(* CoDeSys 2.3 library: EmsUdp2Lcc.lib *)
(* Libraries: SysLibSem.lib 7.1.13 17:20:52, Standard.LIB 4.10.05 12:14:46 *)

(* Global variable list: EmsDrv_Global *)
VAR_GLOBAL
    bEmsOK : BOOL;
    bPreEmsOK : BOOL;
    lastEmsBild : INT := -1;

	dwEmsFifoOut: ARRAY[0..255] OF DWORD;
	bEmsFifoOutWrIndex: BYTE;
	bEmsFifoOutRdIndex: BYTE;
	bEmsFifoOutCount:BYTE;
    cntFifoOutFull : DWORD := 0;
    cntFifoOutBusy : DWORD := 0;
    hndFifoOutSema : DWORD := 0;
    cntFifoOutSemaErr : DWORD := 0;
    cntFifoOutSemaIni : DWORD := 0;

	dwEmsFifoIn: ARRAY[0..255] OF DWORD;
	bEmsFifoInWrIndex: BYTE;
	bEmsFifoInRdIndex: BYTE;
	bEmsFifoInCount:BYTE;

	EmsBild:ARRAY [1..30] OF BOOL;
	InEms: DWORD := 0;

    byToggle : BYTE;
END_VAR

VAR_GLOBAL RETAIN PERSISTENT
	bRunWithEMS: BOOL;
    bEnableEmsScaling: BOOL;

    bDummy: BOOL;

	iEmsAktBild:INT;


	rKatzMetRef: REAL;
	rHeigMetRef: REAL;
	rSlewMetRef: REAL;
	rAneoMetRef: REAL;
	rTrimMetRef: REAL;
	rLastMetRef: REAL;
	rSkewMetRef: REAL;
	rTravMetRef: REAL;
	rListMetRef: REAL;
	rKatzMetMax: REAL;
	rHeigMetMax: REAL;
	rSlewMetMax: REAL;
	rAneoMetMax: REAL;
	rTrimMetMax: REAL;
	rLastMetMax: REAL;
	rSkewMetMax: REAL;
	rTravMetMax: REAL;
	rListMetMax: REAL;
	rKatzMetMin: REAL;
	rHeigMetMin: REAL;
	rSlewMetMin: REAL;
	rAneoMetMin: REAL;
	rTrimMetMin: REAL;
	rLastMetMin: REAL;
	rSkewMetMin: REAL;
	rTravMetMin: REAL;
	rListMetMin: REAL;

	diKatzAdc:    DINT;
	diHeigAdc:    DINT;
	diSlewAdc:    DINT;
	diAneoAdc:    DINT;
	diTrimAdc:    DINT;
	diLastAdc:    DINT;
	diSkewAdc:    DINT;
	diTravAdc:    DINT;
	diListAdc:    DINT;
	diKatzAdcMax: DINT;
	diHeigAdcMax: DINT;
	diSlewAdcMax: DINT;
	diAneoAdcMax: DINT;
	diTrimAdcMax: DINT;
	diLastAdcMax: DINT;
	diSkewAdcMax: DINT;
	diTravAdcMax: DINT;
	diListAdcMax: DINT;
	diKatzAdcMin: DINT;
	diHeigAdcMin: DINT;
	diSlewAdcMin: DINT;
	diAneoAdcMin: DINT;
	diTrimAdcMin: DINT;
	diLastAdcMin: DINT;
	diSkewAdcMin: DINT;
	diTravAdcMin: DINT;
	diListAdcMin: DINT;

    StackData:  DWORD;

	bSendToEmsOnlyIfChanged:BOOL:=FALSE;
END_VAR

(* Data type *)
TYPE tEMS_ANEO_DIM:
(
	IBSK_ANEO_KMH       		:=16#0000,  (* Einheit des Windsensors in km/h *)
	IBSK_ANEO_MPH       		:=16#0001,  (* Einheit des Windsensors in mph  *)
	IBSK_ANEO_MS        		:=16#0002   (* Einheit des Windsensors in m/s  *)
);
END_TYPE

(* Data type *)
TYPE tEMS_FLIP:
(
	IBSK_FLIP_WL          			 :=16#01,  (* LB Flipper water side left  (down) *)
	IBSK_FLIP_WR          			 :=16#02,  (* LB Flipper water side right (down) *)
	IBSK_FLIP_LR          			 :=16#04,  (* LB Flipper land  side right (down) *)
	IBSK_FLIP_LL          			 :=16#08   (* LB Flipper land  side left  (down) *)
);
END_TYPE

(* Data type *)
TYPE tEMS_IBSK :
(
	IBSK_STEUER       := 0,         (* DB1 = Checksumme über 4-ByteEinheit, DB2 und DB3 = Steuerbezeichnung *)

	IBSK_KATZ_MET     := 101,       (* Float in Meter  *)   (* Meterwert des Antriebes *)
	IBSK_HEIG_MET     := 102,       (* Float in Meter  *)
	IBSK_SLEW_MET     := 103,       (* Float in Grad   *)
	IBSK_ANEO_MET     := 104,       (* Float in m/s    *)
	IBSK_TRIM_MET     := 105,       (* Float in Grad   *)
	IBSK_LAST_MET     := 106,       (* Float in Tonnen *)
	IBSK_SKEW_MET     := 107,       (* Float in Grad   *)
	IBSK_TRAV_MET     := 108,       (* Float in Meter  *)
	IBSK_LIST_MET     := 109,       (* Float in Grad   *)

	IBSK_KATZ_MET_REF := 111,       (* Float *)  (* Refernzwerte der Antriebes *)
	IBSK_HEIG_MET_REF := 112,       (* Float *)
	IBSK_SLEW_MET_REF := 113,       (* Float *)
	IBSK_ANEO_MET_REF := 114,       (* Float *)
	IBSK_TRIM_MET_REF := 115,       (* Float *)
	IBSK_LAST_MET_REF := 116,       (* Float *)
	IBSK_SKEW_MET_REF := 117,       (* Float *)
	IBSK_TRAV_MET_REF := 118,       (* Float *)
	IBSK_LIST_MET_REF := 119,       (* Float *)

 	IBSK_KATZ_ADC     := 121,       (* Integer in Digit von -4096 bis +4095 *)   (* analogwert des Antriebes *)
	IBSK_HEIG_ADC     := 122,       (* Integer in Digit von -4096 bis +4095 *)
	IBSK_SLEW_ADC     := 123,       (* Integer in Digit von -4096 bis +4095 *)
	IBSK_ANEO_ADC     := 124,       (* Integer in Digit von -4096 bis +4095 *)
	IBSK_TRIM_ADC     := 125,       (* Integer in Digit von -4096 bis +4095 *)
	IBSK_LAST_ADC     := 126,       (* Integer in Digit von -4096 bis +4095 *)
	IBSK_SKEW_ADC     := 127,       (* Integer in Digit von -4096 bis +4095 *)
	IBSK_TRAV_ADC     := 128,       (* Integer in Digit von -4096 bis +4095 *)
	IBSK_LIST_ADC     := 129,       (* Integer in Digit von -4096 bis +4095 *)

	IBSK_NORTH_DIR    := 130,       (* Integer *)   (* Nordrichtung in Grad bezueglich Kran vorne (Boom) *)
	IBSK_KATZ_DIR     := 131,       (* Integer *)   (* Bewegungsrichtung des Antriebes *)
	IBSK_HEIG_DIR     := 132,       (* Integer *)   (* wird noch ignoriert *)
	IBSK_SLEW_DIR     := 133,       (* Integer *)
	IBSK_ANEO_DIR     := 134,       (* Integer *)   (* Windrichtung in Grad bezueglich Kran vorne (Boom) *)
	IBSK_TRIM_DIR     := 135,       (* Integer *)
	IBSK_LAST_DIR     := 136,       (* Integer *)
	IBSK_SKEW_DIR     := 137,       (* Integer *)
	IBSK_TRAV_DIR     := 138,       (* Integer *)
	IBSK_LIST_DIR     := 139,       (* Integer *)

	IBSK_STEU_EIN     := 140,       (* Integer 1=An, 0=Aus *)   (* für Maschinendatenerfassung *)
	IBSK_KATZ_EIN     := 141,       (* Integer 1=An, 0=Aus *)
	IBSK_HEIG_EIN     := 142,       (* Integer 1=An, 0=Aus *)
	IBSK_SLEW_EIN     := 143,       (* Integer 1=An, 0=Aus *)
	IBSK_TRIM_EIN     := 145,       (* Integer 1=An, 0=Aus *)
	IBSK_SKEW_EIN     := 147,       (* Integer 1=An, 0=Aus *)
	IBSK_TRAV_EIN     := 148,       (* Integer 1=An, 0=Aus *)
	IBSK_LIST_EIN     := 149,       (* Integer 1=An, 0=Aus *)

	IBSK_KATZ_MET_MAX := 151,       (* Float in Meter  *)
	IBSK_HEIG_MET_MAX := 152,       (* Float in Meter  *)
	IBSK_SLEW_MET_MAX := 153,       (* Float in Grad   *)
	IBSK_ANEO_MET_MAX := 154,       (* Float in m/s    *)
	IBSK_TRIM_MET_MAX := 155,       (* Float in Grad   *)
	IBSK_LAST_MET_MAX := 156,       (* Float in Tonnen *)
	IBSK_SKEW_MET_MAX := 157,       (* Float in Grad   *)
	IBSK_TRAV_MET_MAX := 158,       (* Float in Meter  *)
	IBSK_LIST_MET_MAX := 159,       (* Float in Grad   *)

	IBSK_KATZ_MET_MIN := 161,       (* Float in Meter  *)
	IBSK_HEIG_MET_MIN := 162,       (* Float in Meter  *)
	IBSK_SLEW_MET_MIN := 163,       (* Float in Grad   *)
	IBSK_ANEO_MET_MIN := 164,       (* Float in m/s    *)
	IBSK_TRIM_MET_MIN := 165,       (* Float in Grad   *)
	IBSK_LAST_MET_MIN := 166,       (* Float in Tonnen *)
	IBSK_SKEW_MET_MIN := 167,       (* Float in Grad   *)
	IBSK_TRAV_MET_MIN := 168,       (* Float in Meter  *)
	IBSK_LIST_MET_MIN := 169,       (* Float in Grad   *)

	IBSK_KATZ_ADC_MAX := 171,       (* Integer in digit von -4096 bis 4095 *)
	IBSK_HEIG_ADC_MAX := 172,       (* Integer *)
	IBSK_SLEW_ADC_MAX := 173,       (* Integer *)
	IBSK_ANEO_ADC_MAX := 174,       (* Integer *)
	IBSK_TRIM_ADC_MAX := 175,       (* Integer *)
	IBSK_LAST_ADC_MAX := 176,       (* Integer *)
	IBSK_SKEW_ADC_MAX := 177,       (* Integer *)
	IBSK_TRAV_ADC_MAX := 178,       (* Integer *)
	IBSK_LIST_ADC_MAX := 179,       (* Integer *)

	IBSK_KATZ_ADC_MIN := 181,       (* Integer in digit von -4096 bis 4095 *)
	IBSK_HEIG_ADC_MIN := 182,       (* Integer in digit *)
	IBSK_SLEW_ADC_MIN := 183,       (* Integer in digit *)
	IBSK_ANEO_ADC_MIN := 184,       (* Integer in digit *)
	IBSK_TRIM_ADC_MIN := 185,       (* Integer in digit *)
	IBSK_LAST_ADC_MIN := 186,       (* Integer in digit *)
	IBSK_SKEW_ADC_MIN := 187,       (* Integer in digit *)
	IBSK_TRAV_ADC_MIN := 188,       (* Integer in digit *)
	IBSK_LIST_ADC_MIN := 189,       (* Integer in digit *)

	IBSK_BOOM_INFO    := 196,       (* Integer mit Bitbeutung *)
                                    (* 16#0001 = YES "LS1 Boom Up Activated"  *)
                                    (* 16#0002 = YES "LS2 Boom Up Activated"  *)
                                    (* 16#0004 = YES "Slack Rope Left"        *)
                                    (* 16#0008 = YES "Slack Rope Right"       *)
                                    (* 16#0010 = YES "Hook Open"              *)
                                    (* 16#0020 = YES "Hook Closed"            *)
                                    (* 16#0040 = YES "Boom Locked"            *)
                                    (* 16#0080 = YES "LS > 70° Boom Position" *)
                                    (* 16#0100 = YES "In Locking Zone"        *)
                                    (* 16#0200 = YES "LS Boom Down Activated" *)

	IBSK_BOOM_MET  	  := 197,       (* Float in Grad *)
	IBSK_SPRE_MET     := 198,       (* Float in feet *)

	IBSK_FLIP_TWIN    := 199,       (* Integer LB = Flipper und HB = Twin-Lift *)

                                    (* Funktionsbeschreibung am Spreadder *)
                                    (* FLIP = flipper    *)
                                    (* TWIN = twin-lift  *)
                                    (* LOCK = twist-lock *)
                                    (* PROB = probe-pin = deposition point *)

                                    (* Positionsbeschreibung am Spreadder *)
                                    (* zuert water- oder land-side *)
                                    (* dann left oder right *)
                                    (* w = water side *)
                                    (* l = land  side *)
                                    (* l = left       *)
                                    (* r = right      *)
                                    (* t = twin lift  *)


	IBSK_LOCK_PROB    := 200,       (* Integer twist locks und probe pin *)



	IBSK_ANEO_EINHEIT := 201,       (* Integer *) (* Einheit für den Windsensor *)

	IBSK_X_POS        := 204,       (* Integer *) (* Containerposition *)
	IBSK_Y_POS        := 205,       (* Integer *) (* Containerposition *)
	IBSK_Z_POS        := 206,       (* Integer *) (* Containerposition *)
	IBSK_X_DIR        := 207,       (* Zeichen *) (* +,-,* (entspricht: 1,2,3) *)
	IBSK_Y_DIR        := 208,       (* Zeichen *) (* +,-,* (entspricht: 1,2,3) *)
	IBSK_Z_DIR        := 209,       (* Zeichen *) (* +,-,* (entspricht: 1,2,3) *)

	IBSK_ERROR_SET    := 210,       (* Integer Fehler  setzten *)
	IBSK_ERROR_CLEAR  := 211,       (* Integer Fehler  löschen *)
	IBSK_WARN_SET     := 212,       (* Integer Warnung setzten *)
	IBSK_WARN_CLEAR   := 213,       (* Integer Warnung löschen *)

    IBSK_SPRE2_MET    := 215,       (* Tandemspreader Spreader 2: Float in feet *)
    IBSK_FLIP2_TWIN2  := 216,       (* Tandemspreader Spreader 2: Integer LB = Flipper und HB = Twin-Lift *)
    IBSK_LOCK2_PROB2  := 217,       (* Tandemspreader Spreader 2: Integer twist locks und probe pin *)

	IBSK_BILD         := 220,       (* Integer Bildnummer *)
                                    (*  1 = BILD1                        *)
                                    (*  2 = BILD2                        *)
                                    (*  3 = BILD3                        *)
                                    (*  4 = BILD4                        *)
                                    (*  5 = SCALierbild                  *)
                                    (*  6 = Menübild                     *)
                                    (* 10 = COM2-Testbild                *)
                                    (* 11 = Maschinendatenbild 1         *)
                                    (* 12 = Maschinendatenbild 2         *)
                                    (* 13 = Maschinendatenbild 3         *)
                                    (* 14 = Langzeitmaschinendatenbild 1 *)
                                    (* 15 = Langzeitmaschinendatenbild 2 *)
                                    (* 16 = Langzeitmaschinendatenbild 3 *)
                                    (* 19 = zuletzt angewähltes Bild     *)
                                    (*      der Bilder 1 bis 6           *)
                                    (* 26 = BILD neu zeichnen            *)
                                    (* 27 = IBS-Testbild                 *)
                                    (* 28 = BILD5                        *)
                                    (* 29 = BILD6                        *)
                                    (* 30 = BILD_BOOM                    *)

	IBSK_TAST         := 221,       (* Integer HB = Taste  *)
                                    (* TAS_B4 =  1 *)
                                    (* TAS_CL =  2 *)
                                    (* TAS_B5 =  3 *)
                                    (* TAS_EN =  4 *)
                                    (* TAS_B6 =  5 *)
                                    (* TAS_KE =  6 *)
                                    (* TAS_B7 =  7 *)
                                    (* TAS_LI =  9 *)
                                    (* TAS_B1 = 10 *)
                                    (* TAS_RE = 11 *)
                                    (* TAS_B2 = 12 *)
                                    (* TAS_HO = 13 *)
                                    (* TAS_B3 = 14 *)
                                    (* TAS_AB = 15 *)
                                    (*        LB = Repeat *)
                                    (* 1 <= Repeat <= 255 *)
	IBSK_NEW_COM_MODE := 230,	    (* Integer Umschalten in neuen Kommunikationsmode *)
									(* keine Wandlung von Floats *)
							    	(* Schreiben zum EMS: Daten bleiben stehen, bis neue Daten gesendet werden *)
									(* Lesen von EMS: Auswertung von Daten nur bei Änderung *)

    IBSK_STACK_DATA   := 231,       (* Stackdaten DWORD (4 BYTE) *)
                                    (* -> IBS-Kennung, Daten-Kennung, Stack-Nr, Wert *)

    IBSK_MDE2_DATA    := 232,       (* Maschinendaten Bild2 DWORD (4 BYTE) *)
                                    (* -> IBS-Kennung, Daten-Kennung, WORD-Wert *)
    IBSK_MDE3_DATA    := 233,       (* Maschinendaten Bild3 DWORD (4 BYTE) *)
                                    (* -> IBS-Kennung, Daten-Kennung, WORD-Wert *)

	IBSK_GPS_DELTAY   := 234,		(* Abweichung des Krans von der Stackfahrspur *)
	IBSK_GPS_ANGLE    := 235,		(* Winkel des Krans gegenüber der Stackfahrspur *)
	IBSK_GPS_STEERDIR := 236,		(* Lenkrichtung, um zurück auf did Stackfahrspur zu kommen *)

    IBSK_EMS_MODE     := 237        (* EMS-Modus ; Spezielle/Kundenspezifische Anpassungen *)
                                    (* z.Zt.: 0x01 - IBSK_EMS_MODE_MASK_XYZ_2CHAR *) (* 12.01.04 V2.50        *)
                                    (*        0x02 - IBSK_EMS_MODE_MASK_B3_CUST1  *) (* 12.01.04 V2.50        *)
                                    (*        0x04 - IBSK_EMS_MODE_MASK_YZ_2CHAR  *) (* 13.03.09 V2.55 IR1745 *)
                                    (*        0x08 - IBSK_EMS_MODE_MASK_STACK_BIN *) (* 17.02.11 V2.56 RT188  *)
                                    (*        0x80 - IBSK_EMS_MODE_MASK_SET       *)

);
END_TYPE

(* Data type *)
TYPE tEMS_LOCK:
(
	IBSK_LOCK_WL          		 :=16#01,  (* LB Twist lock           water side left  (locked)  *)
	IBSK_LOCK_WR          		 :=16#02,  (* LB Twist lock           water side right (locked)  *)
	IBSK_LOCK_LR          		 :=16#04,  (* LB Twist lock           land  side left  (locked)  *)
	IBSK_LOCK_LL          		 :=16#08,  (* LB Twist lock           land  side right (locked)  *)
	IBSK_LOCK_TWL         		 :=16#10,  (* LB Twist lock twin lift water side left  (locked)  *)
	IBSK_LOCK_TWR         		 :=16#20,  (* LB Twist lock twin lift water side right (locked)  *)
	IBSK_LOCK_TLR         		 :=16#40,  (* LB Twist lock twin lift land  side left  (locked)  *)
	IBSK_LOCK_TLL         		 :=16#80   (* LB Twist lock twin lift land  side right (locked)  *)
);
END_TYPE

(* Data type *)
TYPE tEMS_MDE2 :
(
	IBSK_MDE2K_UNDEF :=0,    (* Undefiniert *)

	IBSK_MDE2K_STEU_AN_1,    (* Kurzzeitspeicher Steuerung An (Anzahl)   1. WORD *)
	IBSK_MDE2K_STEU_AN_2,    (* Kurzzeitspeicher Steuerung An (Anzahl)   2. WORD *)
	IBSK_MDE2K_STEU_ZEIT_1,  (* Kurzzeitspeicher Steuerung An (Dauer)    1. WORD *)
	IBSK_MDE2K_STEU_ZEIT_2,  (* Kurzzeitspeicher Steuerung An (Dauer)    2. WORD *)
	IBSK_MDE2K_KATZ_AN_1,    (* Kurzzeitspeicher Katzantrieb An (Anzahl) 1. WORD *)
	IBSK_MDE2K_KATZ_AN_2,    (* Kurzzeitspeicher Katzantrieb An (Anzahl) 2. WORD *)
	IBSK_MDE2K_KATZ_ZEIT_1,  (* Kurzzeitspeicher Katzantrieb An (Dauer)  1. WORD *)
	IBSK_MDE2K_KATZ_ZEIT_2,  (* Kurzzeitspeicher Katzantrieb An (Dauer)  2. WORD *)
	IBSK_MDE2K_DREH_AN_1,    (* Kurzzeitspeicher Drehantrieb An (Anzahl) 1. WORD *)
	IBSK_MDE2K_DREH_AN_2,    (* Kurzzeitspeicher Drehantrieb An (Anzahl) 2. WORD *)
	IBSK_MDE2K_DREH_ZEIT_1,  (* Kurzzeitspeicher Drehantrieb An (Dauer)  1. WORD *)
	IBSK_MDE2K_DREH_ZEIT_2,  (* Kurzzeitspeicher Drehantrieb An (Dauer)  2. WORD *)
	IBSK_MDE2K_HUB_AN_1,     (* Kurzzeitspeicher Hubantrieb An (Anzahl)  1. WORD *)
	IBSK_MDE2K_HUB_AN_2,     (* Kurzzeitspeicher Hubantrieb An (Anzahl)  2. WORD *)
	IBSK_MDE2K_HUB_ZEIT_1,   (* Kurzzeitspeicher Hubantrieb An (Dauer)   1. WORD *)
	IBSK_MDE2K_HUB_ZEIT_2,   (* Kurzzeitspeicher Hubantrieb An (Dauer)   2. WORD *)
	IBSK_MDE2K_FAHR_AN_1,    (* Kurzzeitspeicher Fahrantrieb An (Anzahl) 1. WORD *)
	IBSK_MDE2K_FAHR_AN_2,    (* Kurzzeitspeicher Fahrantrieb An (Anzahl) 2. WORD *)
	IBSK_MDE2K_FAHR_ZEIT_1,  (* Kurzzeitspeicher Fahrantrieb An (Dauer)  1. WORD *)
	IBSK_MDE2K_FAHR_ZEIT_2,  (* Kurzzeitspeicher Fahrantrieb An (Dauer)  2. WORD *)

	IBSK_MDE2L_STEU_AN_1,    (* Langzeitspeicher Steuerung An (Anzahl)   1. WORD *)
	IBSK_MDE2L_STEU_AN_2,    (* Langzeitspeicher Steuerung An (Anzahl)   2. WORD *)
	IBSK_MDE2L_STEU_ZEIT_1,  (* Langzeitspeicher Steuerung An (Dauer)    1. WORD *)
	IBSK_MDE2L_STEU_ZEIT_2,  (* Langzeitspeicher Steuerung An (Dauer)    2. WORD *)
	IBSK_MDE2L_KATZ_AN_1,    (* Langzeitspeicher Katzantrieb An (Anzahl) 1. WORD *)
	IBSK_MDE2L_KATZ_AN_2,    (* Langzeitspeicher Katzantrieb An (Anzahl) 2. WORD *)
	IBSK_MDE2L_KATZ_ZEIT_1,  (* Langzeitspeicher Katzantrieb An (Dauer)  1. WORD *)
	IBSK_MDE2L_KATZ_ZEIT_2,  (* Langzeitspeicher Katzantrieb An (Dauer)  2. WORD *)
	IBSK_MDE2L_DREH_AN_1,    (* Langzeitspeicher Drehantrieb An (Anzahl) 1. WORD *)
	IBSK_MDE2L_DREH_AN_2,    (* Langzeitspeicher Drehantrieb An (Anzahl) 2. WORD *)
	IBSK_MDE2L_DREH_ZEIT_1,  (* Langzeitspeicher Drehantrieb An (Dauer)  1. WORD *)
	IBSK_MDE2L_DREH_ZEIT_2,  (* Langzeitspeicher Drehantrieb An (Dauer)  2. WORD *)
	IBSK_MDE2L_HUB_AN_1,     (* Langzeitspeicher Hubantrieb An (Anzahl)  1. WORD *)
	IBSK_MDE2L_HUB_AN_2,     (* Langzeitspeicher Hubantrieb An (Anzahl)  2. WORD *)
	IBSK_MDE2L_HUB_ZEIT_1,   (* Langzeitspeicher Hubantrieb An (Dauer)   1. WORD *)
	IBSK_MDE2L_HUB_ZEIT_2,   (* Langzeitspeicher Hubantrieb An (Dauer)   2. WORD *)
	IBSK_MDE2L_FAHR_AN_1,    (* Langzeitspeicher Fahrantrieb An (Anzahl) 1. WORD *)
	IBSK_MDE2L_FAHR_AN_2,    (* Langzeitspeicher Fahrantrieb An (Anzahl) 2. WORD *)
	IBSK_MDE2L_FAHR_ZEIT_1,  (* Langzeitspeicher Fahrantrieb An (Dauer)  1. WORD *)
	IBSK_MDE2L_FAHR_ZEIT_2,  (* Langzeitspeicher Fahrantrieb An (Dauer)  2. WORD *)

	IBSK_MDE2K_LOESCH_1,     (* Kurzzeitspeicher letzte Loeschzeit       1. WORD *)
	IBSK_MDE2K_LOESCH_2,     (* Kurzzeitspeicher letzte Loeschzeit       2. WORD *)

	IBSK_MDE2L_LOESCH_1,     (* Langzeitspeicher letzte Loeschzeit       1. WORD *)
	IBSK_MDE2L_LOESCH_2      (* Langzeitspeicher letzte Loeschzeit       2. WORD *)
);
END_TYPE

(* Data type *)
TYPE tEMS_MDE3 :
(
	IBSK_MDE3K_UNDEF :=0,    (* Undefiniert *)

	IBSK_MDE3K_BIS10_1,      (* Kurzzeitspeicher Last bis 10%       1. WORD *)
	IBSK_MDE3K_BIS10_2,      (* Kurzzeitspeicher Last bis 10%       2. WORD *)
	IBSK_MDE3K_BIS33_1,      (* Kurzzeitspeicher Last bis 33%       1. WORD *)
	IBSK_MDE3K_BIS33_2,      (* Kurzzeitspeicher Last bis 33%       2. WORD *)
	IBSK_MDE3K_BIS66_1,      (* Kurzzeitspeicher Last bis 66%       1. WORD *)
	IBSK_MDE3K_BIS66_2,      (* Kurzzeitspeicher Last bis 66%       2. WORD *)
	IBSK_MDE3K_BIS100_1,     (* Kurzzeitspeicher Last bis 100%      1. WORD *)
	IBSK_MDE3K_BIS100_2,     (* Kurzzeitspeicher Last bis 100%      2. WORD *)
	IBSK_MDE3K_AB100_1,      (* Kurzzeitspeicher Last ueber 100%    1. WORD *)
	IBSK_MDE3K_AB100_2,      (* Kurzzeitspeicher Last ueber 100%    2. WORD *)

	IBSK_MDE3L_BIS10_1,      (* Langzeitspeicher Last bis 10%       1. WORD *)
	IBSK_MDE3L_BIS10_2,      (* Langzeitspeicher Last bis 10%       2. WORD *)
	IBSK_MDE3L_BIS33_1,      (* Langzeitspeicher Last bis 33%       1. WORD *)
	IBSK_MDE3L_BIS33_2,      (* Langzeitspeicher Last bis 33%       2. WORD *)
	IBSK_MDE3L_BIS66_1,      (* Langzeitspeicher Last bis 66%       1. WORD *)
	IBSK_MDE3L_BIS66_2,      (* Langzeitspeicher Last bis 66%       2. WORD *)
	IBSK_MDE3L_BIS100_1,     (* Langzeitspeicher Last bis 100%      1. WORD *)
	IBSK_MDE3L_BIS100_2,     (* Langzeitspeicher Last bis 100%      2. WORD *)
	IBSK_MDE3L_AB100_1,      (* Langzeitspeicher Last ueber 100%    1. WORD *)
	IBSK_MDE3L_AB100_2,      (* Langzeitspeicher Last ueber 100%    2. WORD *)

	IBSK_MDE3K_LOESCH_1,     (* Kurzzeitspeicher letzte Loeschzeit  1. WORD *)
	IBSK_MDE3K_LOESCH_2,     (* Kurzzeitspeicher letzte Loeschzeit  2. WORD *)

	IBSK_MDE3L_LOESCH_1,     (* Langzeitspeicher letzte Loeschzeit  1. WORD *)
	IBSK_MDE3L_LOESCH_2      (* Langzeitspeicher letzte Loeschzeit  2. WORD *)
);
END_TYPE

(* Data type *)
TYPE tEMS_MODE :
(
  (* EMS-Modus ; Spezielle/Kundenspezifische Anpassungen (fuer Interbuskennung IBSK_EMS_MODE := 237) *)
  IBSK_EMS_MODE_MASK_SET       := 16#80,  (* EMS_MODE_MASK_... gesetzt *)
  IBSK_EMS_MODE_MASK_XYZ_2CHAR := 16#01,  (* 12.01.04 V2.50        *)
  IBSK_EMS_MODE_MASK_B3_CUST1  := 16#02,  (* 12.01.04 V2.50        *)
  IBSK_EMS_MODE_MASK_YZ_2CHAR  := 16#04,  (* 13.03.09 V2.55 IR1745 *)
  IBSK_EMS_MODE_MASK_STACK_BIN := 16#08   (* 17.02.11 V2.56 RT188  *)
);
END_TYPE

(* Data type *)
TYPE tEMS_PROBE:
(
	IBSK_PROB_WL          		 :=16#01,  (* HB Probe pin            water side left  (pressed) *)
	IBSK_PROB_WR          		 :=16#02,  (* HB Probe pin            water side right (pressed) *)
	IBSK_PROB_LR          		 :=16#04,  (* HB Probe pin            land  side left  (pressed) *)
	IBSK_PROB_LL          		 :=16#08,  (* HB Probe pin            land  side right (pressed) *)
	IBSK_PROB_TWL         		 :=16#10,  (* HB Probe pin  twin lift water side left  (pressed) *)
	IBSK_PROB_TWR         		 :=16#20,  (* HB Probe pin  twin lift water side right (pressed) *)
	IBSK_PROB_TLR         		 :=16#40,  (* HB Probe pin  twin lift land  side left  (pressed) *)
	IBSK_PROB_TLL         		 :=16#80   (* HB Probe pin  twin lift land  side right (pressed) *)
);
END_TYPE

(* Data type *)
TYPE tEMS_STACK :
(
	IBSK_STACK_UNDEF :=0,  (* Undefiniert *)
	IBSK_STACK_SIZEX,      (* Stacklaenge Travel in 10ft-Einheiten *)
	IBSK_STACK_SIZEY,      (* Stackbreite Trolley in Container-Einheiten *)
	IBSK_STACK_SIZEZ,      (* Stacklaenge Hoist in Container-Einheiten *)
	IBSK_STACK_AKTNR,      (* Aktuelle Stacknummer *)
	IBSK_STACK_NAME0,      (* Stackname 1. Char *)
	IBSK_STACK_NAME1,      (* Stackname 2. Char *)
	IBSK_STACK_DIRROW,     (* Stackausrichtung  Row - Trolley *)
	IBSK_STACK_LABELY,     (* Bezeichnung der Stack-Y-Richtung *)
	IBSK_STACK_FIRST,      (* Position des ersten Containers speichern *)
	IBSK_STACK_LAST,       (* Position des letzten Containers speichern *)
    IBSK_STACK_LABELZ,     (* Bezeichnung der Stack-Z-Richtung *)
	IBSK_STACK_DIRCOL,     (* Stackausrichtung  Column - Travel *)
    IBSK_STACK_FIRST_X1,   (* 1. BYTE des float-Werts der X-Position des ersten Containers *)
    IBSK_STACK_FIRST_X2,   (* 2. BYTE des float-Werts der X-Position des ersten Containers *)
    IBSK_STACK_FIRST_X3,   (* 3. BYTE des float-Werts der X-Position des ersten Containers *)
    IBSK_STACK_FIRST_Y1,   (* 1. BYTE des float-Werts der Y-Position des ersten Containers *)
    IBSK_STACK_FIRST_Y2,   (* 2. BYTE des float-Werts der Y-Position des ersten Containers *)
    IBSK_STACK_FIRST_Y3,   (* 3. BYTE des float-Werts der Y-Position des ersten Containers *)
    IBSK_STACK_LAST_X1,    (* 1. BYTE des float-Werts der X-Position des letzten Containers *)
    IBSK_STACK_LAST_X2,    (* 2. BYTE des float-Werts der X-Position des letzten Containers *)
    IBSK_STACK_LAST_X3,    (* 3. BYTE des float-Werts der X-Position des letzten Containers *)
    IBSK_STACK_LAST_Y1,    (* 1. BYTE des float-Werts der Y-Position des letzten Containers *)
    IBSK_STACK_LAST_Y2,    (* 2. BYTE des float-Werts der Y-Position des letzten Containers *)
    IBSK_STACK_LAST_Y3,    (* 3. BYTE des float-Werts der Y-Position des letzten Containers *)
    IBSK_STACK_AKT_X1,     (* 1. BYTE des float-Werts der aktuellen X-Position *)
    IBSK_STACK_AKT_X2,     (* 2. BYTE des float-Werts der aktuellen X-Position *)
    IBSK_STACK_AKT_X3,     (* 3. BYTE des float-Werts der aktuellen X-Position *)
    IBSK_STACK_AKT_Y1,     (* 1. BYTE des float-Werts der aktuellen Y-Position *)
    IBSK_STACK_AKT_Y2,     (* 2. BYTE des float-Werts der aktuellen Y-Position *)
    IBSK_STACK_AKT_Y3      (* 3. BYTE des float-Werts der aktuellen Y-Position *)
);
END_TYPE

(* Data type *)
TYPE tEMS_STACK_DATA :
STRUCT
 kenn   : tEMS_STACK;
 nr     : BYTE;
 data   : BYTE;
 toggle : BYTE;
END_STRUCT
END_TYPE

(* Data type *)
TYPE tEMS_TWIN :
(
	IBSK_TWIN             			 :=16#01,  (* HB Twin-lift (aktiv) *)
	IBSK_TANDEM            			 :=16#02,  (* HB Twin-lift (aktiv) *)
	IBSK_ENABLED           			 :=16#04   (* HB Twin-lift (aktiv) *)
);
END_TYPE

(* POU BoomInfoToEms, ST *)
PROGRAM BoomInfoToEms
VAR_INPUT
	Ls1BoomUpActivated: BOOL;
	Ls2BoomUpActivated: BOOL;
	SlackRopeLeft: BOOL;
	SlackRopeRight: BOOL;
	HookOpen: BOOL;
	HookClosed: BOOL;
	BoomLocked: BOOL;
	LsGreater70DegBoomPosition: BOOL;

	InLockingZone: BOOL;
	LsBoomDownActivated: BOOL;
END_VAR
VAR
	pdw: POINTER TO ARRAY[0..3] OF BYTE;
	dwEMSOut: DWORD := 0;
END_VAR
pdw := ADR(dwEMSOut);

pdw^[0] := INT_TO_BYTE(IBSK_LOCK_PROB);
(*pdw^[1] := 0;*)
pdw^[1] := byToggle;
byToggle := byToggle + 1;

pdw^[2].0 := InLockingZone;
pdw^[2].1 := LsBoomDownActivated;


pdw^[3].0 := Ls1BoomUpActivated;
pdw^[3].1 := Ls2BoomUpActivated;
pdw^[3].2 := SlackRopeLeft;
pdw^[3].3 := SlackRopeRight;
pdw^[3].4 := HookOpen;
pdw^[3].5 := HookClosed;
pdw^[3].6 := BoomLocked;
pdw^[3].7 := LsGreater70DegBoomPosition;

EmsOutFifo(dwEMSOut);
END_PROGRAM

(* POU EmsOutFifo, ST *)
FUNCTION EmsOutFifo : BOOL
VAR_INPUT
	dwEmsOut:DWORD;
END_VAR
VAR
 bSemRet : BOOL;
END_VAR
IF( hndFifoOutSema > 0) THEN
 bSemRet := SysSemEnter( hndFifoOutSema);
 IF( bSemRet) THEN

  (* noch Platz im Fifo ?*)
  (*IF (bEmsFifoOutCount <= 255) THEN*)
  IF( bEmsFifoOutCount < 255) THEN
   (*ins Fifo schreiben*)
   dwEmsFifoOut[bEmsFifoOutWrIndex] := dwEmsOut;
   bEmsFifoOutWrIndex := bEmsFifoOutWrIndex+1;
   bEmsFifoOutCount := bEmsFifoOutCount+1;
   EmsOutFifo:=TRUE;
  ELSE
   cntFifoOutFull := cntFifoOutFull + 1;
   EmsOutFifo:=FALSE;
  END_IF

  bSemRet := SysSemLeave( hndFifoOutSema);
  IF( NOT bSemRet) THEN
   cntFifoOutSemaErr := cntFifoOutSemaErr + 1;
  END_IF
 ELSE
  cntFifoOutBusy := cntFifoOutBusy + 1;
 END_IF
ELSE
 cntFifoOutSemaIni := cntFifoOutSemaIni + 1;
END_IF
END_FUNCTION

(* POU EMS_BildUpdate, ST *)
PROGRAM EMS_BildUpdate
VAR
	ii:BYTE;
END_VAR
(* beim Erststart auf Bild1 umschalten *)
IF (iEmsAktBild = -1) THEN
	BildNumToEms(1);

ELSE
	FOR ii:=1 TO 30 BY 1 DO
		IF (EmsBild[ii] = TRUE) THEN
			BildNumToEms(ii);
		END_IF
	END_FOR
END_IF
END_PROGRAM

(* POU BildNumToEms, ST *)
FUNCTION BildNumToEms:BOOL
VAR_INPUT
	Wert: INT;
END_VAR
VAR
	pdw: POINTER TO ARRAY[0..3] OF BYTE;
	pint: POINTER TO ARRAY[0..1] OF BYTE;
	dwEMSOut: DWORD;
END_VAR
pdw := ADR(dwEMSOut);
pint := ADR(Wert);

pdw^[0] := INT_TO_BYTE(IBSK_BILD);
(*pdw^[1] := 0;*)
pdw^[1] := byToggle;
byToggle := byToggle + 1;
pdw^[2] := pint^[1];
pdw^[3] := pint^[0];

BildNumToEms := EmsOutFifo(dwEMSOut);
END_FUNCTION

(* POU EMS_DataInterpreter, ST *)
PROGRAM EMS_DataInterpreter
VAR_INPUT
	bEnable: BOOL;
END_VAR
VAR
	dwEmsIn:DWORD;
	Kennung:tEMS_IBSK;
END_VAR
IF NOT bEnable THEN
	RETURN;
END_IF

IF (bEmsFifoInCount > 0) THEN
	(*aus Fifo lesen *)
	dwEmsIn := dwEmsFifoIn[bEmsFifoInRdIndex];
	bEmsFifoInRdIndex := bEmsFifoInRdIndex+1;
	bEmsFifoInCount := bEmsFifoInCount-1;
	Kennung := GetIbsKennung(dwEmsIn);

	CASE Kennung OF
		IBSK_STEUER:
	;
		IBSK_KATZ_MET,	(* Float in Meter  *)   (* Meterwert des Antriebes *)
		IBSK_HEIG_MET,  (* Float in Meter  *)
		IBSK_SLEW_MET,  (* Float in Grad   *)
		IBSK_ANEO_MET,  (* Float in m/s    *)
		IBSK_TRIM_MET,  (* Float in Grad   *)
		IBSK_LAST_MET,  (* Float in Tonnen *)
		IBSK_SKEW_MET,  (* Float in Grad   *)
		IBSK_TRAV_MET,  (* Float in Meter  *)
		IBSK_LIST_MET:  (* Float in Grad   *)
	;
		IBSK_KATZ_MET_REF:  (* Float *)  (* Refernzwerte der Antriebes *)
			rKatzMetRef := FloatFromEms(dwEmsIn);
		IBSK_HEIG_MET_REF:  (* Float *)
			rHeigMetRef := FloatFromEms(dwEmsIn);
		IBSK_SLEW_MET_REF:  (* Float *)
			rSlewMetRef := FloatFromEms(dwEmsIn);
		IBSK_ANEO_MET_REF:  (* Float *)
			rAneoMetRef := FloatFromEms(dwEmsIn);
		IBSK_TRIM_MET_REF:  (* Float *)
			rTrimMetRef := FloatFromEms(dwEmsIn);
		IBSK_LAST_MET_REF:  (* Float *)
			rLastMetRef := FloatFromEms(dwEmsIn);
		IBSK_SKEW_MET_REF:  (* Float *)
			rSkewMetRef := FloatFromEms(dwEmsIn);
		IBSK_TRAV_MET_REF:  (* Float *)
			rTravMetRef := FloatFromEms(dwEmsIn);
		IBSK_LIST_MET_REF:  (* Float *)
			rListMetRef := FloatFromEms(dwEmsIn);


		IBSK_KATZ_MET_MAX:  (* Float in Meter  *)
			rKatzMetMax := FloatFromEms(dwEmsIn);
		IBSK_HEIG_MET_MAX:  (* Float in Meter  *)
			rHeigMetMax := FloatFromEms(dwEmsIn);
		IBSK_SLEW_MET_MAX:  (* Float in Grad   *)
			rSlewMetMax := FloatFromEms(dwEmsIn);
		IBSK_ANEO_MET_MAX:  (* Float in m/s    *)
			rAneoMetMax := FloatFromEms(dwEmsIn);
		IBSK_TRIM_MET_MAX:  (* Float in Grad   *)
			rTrimMetMax := FloatFromEms(dwEmsIn);
		IBSK_LAST_MET_MAX: (* Float in Tonnen *)
			rLastMetMax := FloatFromEms(dwEmsIn);
		IBSK_SKEW_MET_MAX:  (* Float in Grad   *)
			rSkewMetMax := FloatFromEms(dwEmsIn);
		IBSK_TRAV_MET_MAX:  (* Float in Meter  *)
			rTravMetMax := FloatFromEms(dwEmsIn);
		IBSK_LIST_MET_MAX:  (* Float in Grad   *)
			rListMetMax := FloatFromEms(dwEmsIn);

		IBSK_KATZ_MET_MIN:  (* Float in Meter  *)
			rKatzMetMin := FloatFromEms(dwEmsIn);
		IBSK_HEIG_MET_MIN:  (* Float in Meter  *)
			rHeigMetMin := FloatFromEms(dwEmsIn);
		IBSK_SLEW_MET_MIN:  (* Float in Grad   *)
			rSlewMetMin := FloatFromEms(dwEmsIn);
		IBSK_ANEO_MET_MIN:  (* Float in m/s    *)
			rAneoMetMin := FloatFromEms(dwEmsIn);
		IBSK_TRIM_MET_MIN:  (* Float in Grad   *)
			rTrimMetMin := FloatFromEms(dwEmsIn);
		IBSK_LAST_MET_MIN:  (* Float in Tonnen *)
			rLastMetMin := FloatFromEms(dwEmsIn);
		IBSK_SKEW_MET_MIN:  (* Float in Grad   *)
			rSkewMetMin := FloatFromEms(dwEmsIn);
		IBSK_TRAV_MET_MIN:  (* Float in Meter  *)
			rTravMetMin := FloatFromEms(dwEmsIn);
		IBSK_LIST_MET_MIN:  (* Float in Grad   *)
			rListMetMin := FloatFromEms(dwEmsIn);

	 	IBSK_KATZ_ADC:			(* Integer in Digit von -4096 bis +4095 *)   (* analogwert des Antriebes *)
			diKatzAdc := IntFromEms(dwEmsIn);
		IBSK_HEIG_ADC:  		(* Integer in Digit von -4096 bis +4095 *)
			diHeigAdc := IntFromEms(dwEmsIn);
		IBSK_SLEW_ADC:  		(* Integer in Digit von -4096 bis +4095 *)
			diSlewAdc := IntFromEms(dwEmsIn);
		IBSK_ANEO_ADC:  		(* Integer in Digit von -4096 bis +4095 *)
			diAneoAdc := IntFromEms(dwEmsIn);
		IBSK_TRIM_ADC:			(* Integer in Digit von -4096 bis +4095 *)
			diTrimAdc := IntFromEms(dwEmsIn);
		IBSK_LAST_ADC:  (* Integer in Digit von -4096 bis +4095 *)
			diLastAdc := IntFromEms(dwEmsIn);
		IBSK_SKEW_ADC:  (* Integer in Digit von -4096 bis +4095 *)
			diSkewAdc := IntFromEms(dwEmsIn);
		IBSK_TRAV_ADC:  (* Integer in Digit von -4096 bis +4095 *)
			diTravAdc := IntFromEms(dwEmsIn);
		IBSK_LIST_ADC:  (* Integer in Digit von -4096 bis +4095 *)
			diListAdc := IntFromEms(dwEmsIn);

		IBSK_KATZ_DIR,  (* Integer *)   (* Bewegungsrichtung des Antriebes *)
		IBSK_HEIG_DIR,  (* Integer *)   (* wird noch ignoriert *)
		IBSK_SLEW_DIR,  (* Integer *)
		IBSK_ANEO_DIR,  (* Integer *)
		IBSK_TRIM_DIR,  (* Integer *)
		IBSK_LAST_DIR,  (* Integer *)
		IBSK_SKEW_DIR,  (* Integer *)
		IBSK_TRAV_DIR,  (* Integer *)
		IBSK_LIST_DIR: (* Integer *)
	;
		IBSK_STEU_EIN,  (* Integer 1=An, 0=Aus *)   (* für Maschinendatenerfassung *)
		IBSK_KATZ_EIN,  (* Integer 1=An, 0=Aus *)
		IBSK_HEIG_EIN,  (* Integer 1=An, 0=Aus *)
		IBSK_SLEW_EIN,  (* Integer 1=An, 0=Aus *)
		IBSK_TRIM_EIN,  (* Integer 1=An, 0=Aus *)
		IBSK_SKEW_EIN,  (* Integer 1=An, 0=Aus *)
		IBSK_TRAV_EIN,  (* Integer 1=An, 0=Aus *)
		IBSK_LIST_EIN:  (* Integer 1=An, 0=Aus *)
	;

		IBSK_KATZ_ADC_MAX:  (* Integer in digit von -4096 bis 4095 *)
			diKatzAdcMax := IntFromEms(dwEmsIn);
		IBSK_HEIG_ADC_MAX:  (* Integer *)
			diHeigAdcMax := IntFromEms(dwEmsIn);
		IBSK_SLEW_ADC_MAX:  (* Integer *)
			diSlewAdcMax := IntFromEms(dwEmsIn);
		IBSK_ANEO_ADC_MAX:  (* Integer *)
			diAneoAdcMax := IntFromEms(dwEmsIn);
		IBSK_TRIM_ADC_MAX:  (* Integer *)
			diTrimAdcMax := IntFromEms(dwEmsIn);
		IBSK_LAST_ADC_MAX:  (* Integer *)
			diLastAdcMax := IntFromEms(dwEmsIn);
		IBSK_SKEW_ADC_MAX:  (* Integer *)
			diSkewAdcMax := IntFromEms(dwEmsIn);
		IBSK_TRAV_ADC_MAX:  (* Integer *)
			diTravAdcMax := IntFromEms(dwEmsIn);
		IBSK_LIST_ADC_MAX: (* Integer *)
			diListAdcMax := IntFromEms(dwEmsIn);

		IBSK_KATZ_ADC_MIN:  (* Integer in digit von -4096 bis 4095 *)
			diKatzAdcMin := IntFromEms(dwEmsIn);
		IBSK_HEIG_ADC_MIN:  (* Integer in digit *)
			diHeigAdcMin := IntFromEms(dwEmsIn);
		IBSK_SLEW_ADC_MIN:  (* Integer in digit *)
			diSlewAdcMin := IntFromEms(dwEmsIn);
		IBSK_ANEO_ADC_MIN:  (* Integer in digit *)
			diAneoAdcMin := IntFromEms(dwEmsIn);
		IBSK_TRIM_ADC_MIN:  (* Integer in digit *)
			diTrimAdcMin := IntFromEms(dwEmsIn);
		IBSK_LAST_ADC_MIN:  (* Integer in digit *)
			diLastAdcMin := IntFromEms(dwEmsIn);
		IBSK_SKEW_ADC_MIN:  (* Integer in digit *)
			diSkewAdcMin := IntFromEms(dwEmsIn);
		IBSK_TRAV_ADC_MIN:  (* Integer in digit *)
			diTravAdcMin := IntFromEms(dwEmsIn);
		IBSK_LIST_ADC_MIN:  (* Integer in digit *)
			diListAdcMin := IntFromEms(dwEmsIn);

		IBSK_BOOM_INFO:  (* Integer mit Bitbeutung *)
	                                 (* 16#0001 = YES "LS1 Boom Up Activated"  *)
	                                 (* 16#0002 = YES "LS2 Boom Up Activated"  *)
	                                 (* 16#0004 = YES "Slack Rope Left"        *)
	                                 (* 16#0008 = YES "Slack Rope Right"       *)
	                                 (* 16#0010 = YES "Hook Open"              *)
	                                 (* 16#0020 = YES "Hook Closed"            *)
	                                 (* 16#0040 = YES "Boom Locked"            *)
	                                 (* 16#0080 = YES "LS > 70° Boom Position" *)
	                                 (* 16#0100 = YES "In Locking Zone"        *)
	                                 (* 16#0200 = YES "LS Boom Down Activated" *)
	;
		IBSK_BOOM_MET,  (* Float in Grad *)
		IBSK_SPRE_MET:  (* Float in feet *)
	;
		IBSK_FLIP_TWIN:  (* Integer LB = Flipper und HB = Twin-Lift *)
	;
	                                 (* Funktionsbeschreibung am Spreadder *)
	                                 (* FLIP = flipper    *)
	                                 (* TWIN = twin-lift  *)
	                                 (* LOCK = twist-lock *)
	                                 (* PROB = probe-pin = deposition point *)

	                                    (* Positionsbeschreibung am Spreadder *)
	                                    (* zuert water- oder land-side *)
	                                    (* dann left oder right *)
	                                    (* w = water side *)
	                                    (* l = land  side *)
	                                    (* l = left       *)
	                                    (* r = right      *)
	                                    (* t = twin lift  *)


		IBSK_LOCK_PROB:  (* Integer twist locks und probe pin *)
	;


		IBSK_ANEO_EINHEIT:  (* Integer *) (* Einheit für den Windsensor *)
	;
		IBSK_X_POS,  (* Integer *) (* Containerposition *)
		IBSK_Y_POS,  (* Integer *) (* Containerposition *)
		IBSK_Z_POS,  (* Integer *) (* Containerposition *)
		IBSK_X_DIR,  (* Zeichen *) (* +,-,* *)
		IBSK_Y_DIR,  (* Zeichen *) (* +,-,* *)
		IBSK_Z_DIR:  (* Zeichen *) (* +,-,* *)
	;
		IBSK_ERROR_SET:    (* Integer Fehler  setzten *)
	;
		IBSK_ERROR_CLEAR:  (* Integer Fehler  löschen *)
	;
		IBSK_WARN_SET:     (* Integer Warnung setzten *)
	;
		IBSK_WARN_CLEAR:   (* Integer Warnung löschen *)
	;
		IBSK_BILD: (* Integer Bildnummer *)
			iEmsAktBild := INT_TO_BYTE(IntFromEms(dwEmsIn));
		IBSK_TAST:  (* Integer HB = Taste  *)
	;                                   (* TAS_B4 =  1 *)
	                                    (* TAS_CL =  2 *)
	                                    (* TAS_B5 =  3 *)
	                                    (* TAS_EN =  4 *)
	                                    (* TAS_B6 =  5 *)
	                                    (* TAS_KE =  6 *)
	                                    (* TAS_B7 =  7 *)
	                                    (* TAS_LI =  9 *)
	                                    (* TAS_B1 = 10 *)
	                                    (* TAS_RE = 11 *)
	                                    (* TAS_B2 = 12 *)
	                                    (* TAS_HO = 13 *)
	                                    (* TAS_B3 = 14 *)
	                                    (* TAS_AB = 15 *)
	                                    (*        LB = Repeat *)
	                                    (* 1 <= Repeat <= 255 *)

        IBSK_STACK_DATA:                (* Stackdaten DWORD (4 Byte) *)
            StackData := dwEmsIn;

	END_CASE
END_IF
END_PROGRAM

(* POU GetIbsKennung, ST *)
FUNCTION GetIbsKennung : tEMS_IBSK
VAR_INPUT
	InEMS:DWORD;
END_VAR
VAR
	pdw: POINTER TO ARRAY[0..3] OF BYTE;
END_VAR
pdw := ADR(InEMS);
GetIbsKennung := pdw^[0];
END_FUNCTION

(* POU FloatFromEms, ST *)
FUNCTION FloatFromEms:REAL
VAR_INPUT
	dwEMSIn: DWORD;
END_VAR
VAR
	pdw		: POINTER TO ARRAY[0..3] OF BYTE;
	pWert	: POINTER TO ARRAY[0..3] OF BYTE;
	Wert: REAL;
END_VAR
pdw := ADR(dwEMSIn);
pWert := ADR(Wert);

(* ibs   = mmmmmmmm emmmmmmm seeeeeee kkkkkkkk *)
(* float = seeeeeee emmmmmmm mmmmmmmm mmmmmmmm *)

(* Wert füllen und dabei Bytereihenfolge drehen *)
pWert^[0] := 0;
pWert^[1] := pdw^[3];
pWert^[2] := pdw^[2];
pWert^[3] := pdw^[1];

FloatFromEms := Wert;
END_FUNCTION

(* POU IntFromEms, ST *)
FUNCTION IntFromEms: INT
VAR_INPUT
	dwEMSIn: DWORD;
END_VAR
VAR
	pdw: POINTER TO ARRAY[0..3] OF BYTE;
	pint: POINTER TO ARRAY[0..1] OF BYTE;

	Kennung: tEMS_IBSK;
	Wert: INT;
END_VAR
pdw := ADR(dwEMSIn);
pint := ADR(Wert);

Kennung := pdw^[0];
pint^[1] := pdw^[2];
pint^[0] := pdw^[3];

IntFromEms := Wert;
END_FUNCTION

(* POU EMS_Init, ST *)
PROGRAM EMS_Init

VAR_INPUT
	bEnable:BOOL;
END_VAR

VAR
	bRestart: BOOL := TRUE;
	rtEnable: R_TRIG;
	fbIntToEms:IntToEms;
	Wert:INT;

	Counter: BYTE;
	ton1s: TON;
END_VAR
IF( hndFifoOutSema = 0) THEN
 hndFifoOutSema := SysSemCreate( TRUE);
END_IF

rtEnable( CLK := bEnable);

IF rtEnable.Q THEN
  (* clear FifoOut *)
  bEmsFifoOutCount := 0;
  bEmsFifoOutRdIndex := 0;
  bEmsFifoOutWrIndex := 0;
  (* send New Mode to EMS in both dwords *)
  Counter := 0;
END_IF

ton1s( IN := TRUE, PT := t#1s);

IF ( ton1s.Q = TRUE) AND ( Counter < 5) THEN
  fbIntToEms( Kennung := IBSK_NEW_COM_MODE, Wert := Wert);
  Counter := Counter + 1;
  ton1s( IN := FALSE);
END_IF
END_PROGRAM

(* POU IntToEms, ST *)
FUNCTION_BLOCK IntToEms
VAR_INPUT
	Kennung: tEMS_IBSK;
	Wert: INT;
END_VAR
VAR
	pdw: POINTER TO ARRAY[0..3] OF BYTE;
	pint: POINTER TO ARRAY[0..1] OF BYTE;
	dwEMSOut: DWORD;
	LastdwEMSOut: DWORD;
END_VAR
pdw := ADR(dwEMSOut);
pint := ADR(Wert);

pdw^[0] := INT_TO_BYTE(Kennung);
(*pdw^[1] := 0;*)
pdw^[1] := byToggle;
byToggle := byToggle + 1;
pdw^[2] := pint^[1];
pdw^[3] := pint^[0];

IF bSendToEmsOnlyIfChanged THEN
	IF (LastdwEMSOut <> dwEMSOut) THEN
		EmsOutFifo(dwEMSOut);
	END_IF
ELSE
	EmsOutFifo(dwEMSOut);
END_IF
LastdwEMSOut := dwEMSOut;
END_FUNCTION_BLOCK

(* POU EMS_Mode, ST *)
PROGRAM EMS_Mode

VAR_INPUT
  bEnable : BOOL;
  iWert   : INT;
END_VAR

VAR
  rtEnable : R_TRIG;
  fbIntToEms : IntToEms;

  Counter : BYTE;
  ton1s : TON;
END_VAR
rtEnable( CLK := bEnable);

IF rtEnable.Q THEN
  (* send EMS mode to EMS every second for 5 seconds *)
  Counter := 0;
END_IF

ton1s( IN := TRUE, PT := t#1s);

IF ( ton1s.Q = TRUE) AND ( Counter < 5) THEN
  fbIntToEms( Kennung := IBSK_EMS_MODE, Wert := iWert);
  Counter := Counter + 1;
  ton1s( IN := FALSE);
END_IF
END_PROGRAM

(* POU EMS_Read, ST *)
PROGRAM EMS_Read
VAR_INPUT
	bEnable: BOOL;
	In1: DWORD;
	In2: DWORD;
END_VAR
VAR
	idwEms1Old:DWORD:=0;
	idwEms2Old:DWORD:=0;
END_VAR
IF NOT bEnable OR NOT bRunWithEMS THEN
	RETURN;
END_IF

(* EMS-Daten einlesen *)
IF (In1<>idwEms1Old) THEN
	EmsInFifo(In1);
	idwEms1Old:=In1;
END_IF
IF (In2<>idwEms2Old) THEN
	EmsInFifo(In2);
	idwEms2Old:=In2;
END_IF
END_PROGRAM

(* POU EmsInFifo, ST *)
FUNCTION EmsInFifo : BOOL
VAR_INPUT
	dwEmsIn:DWORD;
END_VAR
VAR
END_VAR
(* noch Platz im Fifo ?*)
IF (bEmsFifoInCount <= 255) THEN
	(*ins Fifo schreiben*)
	 dwEmsFifoIn[bEmsFifoInWrIndex] := dwEmsIn;
	bEmsFifoInWrIndex := bEmsFifoInWrIndex+1;
	bEmsFifoInCount := bEmsFifoInCount+1;
  EmsInFifo:=TRUE;
ELSE
  EmsInFifo:=FALSE;
END_IF
END_FUNCTION

(* POU EMS_Write, ST *)
PROGRAM EMS_Write
VAR_INPUT
  bEnable: BOOL;
END_VAR
VAR_OUTPUT
  Out1: DWORD;
  Out2: DWORD;
END_VAR
VAR
  rtEnable: R_TRIG;
  LastChannel: BYTE := 1;
  bSemRet : BOOL;
END_VAR
rtEnable(CLK:=bEnable);
IF (rtEnable.Q) THEN
	LastChannel := 2;
END_IF

IF NOT bEnable OR NOT bRunWithEMS THEN
	RETURN;
END_IF


IF( hndFifoOutSema > 0) THEN
 bSemRet := SysSemEnter( hndFifoOutSema);
 IF( bSemRet) THEN

  IF (bEmsFifoOutCount>0) THEN
	(* FifoOut-Daten zum EMS senden *)
	IF(LastChannel = 1) THEN
		LastChannel := 2;
	ELSE
		LastChannel := 1;
	END_IF
	IF(LastChannel = 1) THEN
		Out1 := dwEmsFifoOut[bEmsFifoOutRdIndex];
	ELSE
		Out2 := dwEmsFifoOut[bEmsFifoOutRdIndex];
	END_IF
	bEmsFifoOutRdIndex := bEmsFifoOutRdIndex+1;
	bEmsFifoOutCount := bEmsFifoOutCount-1;
  END_IF

  bSemRet := SysSemLeave( hndFifoOutSema);
  IF( NOT bSemRet) THEN
   cntFifoOutSemaErr := cntFifoOutSemaErr + 1;
  END_IF
 ELSE
  cntFifoOutBusy := cntFifoOutBusy + 1;
 END_IF
ELSE
 cntFifoOutSemaIni := cntFifoOutSemaIni + 1;
END_IF
END_PROGRAM

(* POU FlipTwinToEms, ST *)
PROGRAM FlipTwinToEms
VAR_INPUT
	FlipWaterSideLeftDown: BOOL;
	FlipWaterSideRightDown: BOOL;
	FlipLandSideRightDown: BOOL;
	FlipLandSideLeftDown: BOOL;
	TwinLiftActive: BOOL;
END_VAR
VAR_OUTPUT
    FlippersToEMS : WORD;
    TwinToEMS : WORD;
END_VAR
TwinToEMS.0 := TwinLiftActive;

FlippersToEMS.0 := FlipWaterSideLeftDown;
FlippersToEMS.1 := FlipWaterSideRightDown;
FlippersToEMS.2 := FlipLandSideRightDown;
FlippersToEMS.3 := FlipLandSideLeftDown;
END_PROGRAM

(* POU LockProbToEms, ST *)
PROGRAM LockProbToEms
VAR_INPUT
	TlWaterSideLeftLocked: BOOL;
	TlWaterSideRightLocked: BOOL;
	TlLandSideLeftLocked: BOOL;
	TlLandSideRightLocked: BOOL;
	TlTwinLiftWaterSideLeftLocked: BOOL;
	TlTwinLiftWaterSideRightLocked: BOOL;
	TlTwinLiftLandSideLeftLocked: BOOL;
	TlTwinLiftLandSideRightLocked: BOOL;

	PpWaterSideLeftPressed: BOOL;
	PpWaterSideRightPressed: BOOL;
	PpLandSideLeftPressed: BOOL;
	PpLandSideRightPressed: BOOL;
	PpTwinLiftWaterSideLeftPressed: BOOL;
	PpTwinLiftWaterSideRightPressed: BOOL;
	PpTwinLiftLandSideLeftPressed: BOOL;
	PpTwinLiftLandSideRightPressed: BOOL;
END_VAR
VAR_OUTPUT
    TwistlocksToEMS : WORD;
    ProbesToEMS : WORD;
END_VAR
ProbesToEMS.0 := PpWaterSideLeftPressed;
ProbesToEMS.1 := PpWaterSideRightPressed;
ProbesToEMS.2 := PpLandSideRightPressed;
ProbesToEMS.3 := PpLandSideLeftPressed;
ProbesToEMS.4 := PpTwinLiftWaterSideLeftPressed;
ProbesToEMS.5 := PpTwinLiftWaterSideRightPressed;
ProbesToEMS.6 := PpTwinLiftLandSideRightPressed;
ProbesToEMS.7 := PpTwinLiftLandSideLeftPressed;


TwistlocksToEMS.0 := TlWaterSideLeftLocked;
TwistlocksToEMS.1 := TlWaterSideRightLocked;
TwistlocksToEMS.2 := TlLandSideRightLocked;
TwistlocksToEMS.3 := TlLandSideLeftLocked;
TwistlocksToEMS.4 := TlTwinLiftWaterSideLeftLocked;
TwistlocksToEMS.5 := TlTwinLiftWaterSideRightLocked;
TwistlocksToEMS.6 := TlTwinLiftLandSideRightLocked;
TwistlocksToEMS.7 := TlTwinLiftLandSideLeftLocked;
END_PROGRAM

(* POU BuildStackData, ST *)
FUNCTION BuildStackData : tEMS_STACK_DATA
VAR_INPUT
 kenn : tEMS_STACK;
 nr   : BYTE;
 data : BYTE;
END_VAR
VAR
END_VAR
BuildStackData.kenn := kenn;
BuildStackData.nr := nr;
BuildStackData.data := data;
END_FUNCTION

(* POU DirToEms, ST *)
FUNCTION_BLOCK DirToEms
VAR_INPUT
	Kennung: tEMS_IBSK;
	Wert: STRING;
END_VAR
VAR
	pdw: POINTER TO ARRAY[0..3] OF BYTE;
	dwEMSOut: DWORD;
	LastdwEMSOut: DWORD;
END_VAR
(*
Wert: '+' (1) 
Wert: '-' (2)
Wert: '*' (3)
*)
pdw := ADR(dwEMSOut);

pdw^[0] := INT_TO_BYTE(Kennung);
(*pdw^[1] := 0;*)
pdw^[1] := byToggle;
byToggle := byToggle + 1;
pdw^[2] := 0;

IF(Wert='+') THEN pdw^[3] := 1;
ELSIF (Wert='-') THEN pdw^[3] := 2;
ELSIF (Wert='*') THEN pdw^[3] := 3;
END_IF

IF bSendToEmsOnlyIfChanged THEN
	IF (LastdwEMSOut <> dwEMSOut) THEN
		EmsOutFifo(dwEMSOut);
	END_IF
ELSE
	EmsOutFifo(dwEMSOut);
END_IF
LastdwEMSOut := dwEMSOut;
END_FUNCTION_BLOCK

(* POU ErrorClearToEms, ST *)
FUNCTION ErrorClearToEms:BOOL
VAR_INPUT
	Wert: INT;
END_VAR
VAR
	pdw: POINTER TO ARRAY[0..3] OF BYTE;
	pint: POINTER TO ARRAY[0..1] OF BYTE;
	dwEMSOut: DWORD;
END_VAR
pdw := ADR(dwEMSOut);
pint := ADR(Wert);

pdw^[0] := INT_TO_BYTE(IBSK_ERROR_CLEAR);
(*pdw^[1] := 0;*)
pdw^[1] := byToggle;
byToggle := byToggle + 1;

pdw^[2] := pint^[1];
pdw^[3] := pint^[0];

ErrorClearToEms := EmsOutFifo(dwEMSOut);
END_FUNCTION

(* POU ErrorSetToEms, ST *)
FUNCTION ErrorSetToEms:BOOL
VAR_INPUT
	Wert: INT;
END_VAR
VAR
	pdw: POINTER TO ARRAY[0..3] OF BYTE;
	pint: POINTER TO ARRAY[0..1] OF BYTE;
	dwEMSOut: DWORD;
END_VAR
pdw := ADR(dwEMSOut);
pint := ADR(Wert);

pdw^[0] := INT_TO_BYTE(IBSK_ERROR_SET);
(*pdw^[1] := 0;*)
pdw^[1] := byToggle;
byToggle := byToggle + 1;

pdw^[2] := pint^[1];
pdw^[3] := pint^[0];

ErrorSetToEms := EmsOutFifo(dwEMSOut);
END_FUNCTION

(* POU FloatToEms, ST *)
FUNCTION_BLOCK FloatToEms
VAR_INPUT
	Kennung: tEMS_IBSK;
	Wert: REAL;
END_VAR
VAR
	pdw		: POINTER TO ARRAY[0..3] OF BYTE;
	pWert	: POINTER TO ARRAY[0..3] OF BYTE;
	dwEMSOut: DWORD;
	LastdwEMSOut: DWORD;
END_VAR
pdw := ADR(dwEMSOut);
pWert := ADR(Wert);

(* real  = seeeeeee emmmmmmm mmmmmmmm mmmmmmmm *)
(* ibs   = mmmmmmmm emmmmmmm seeeeeee kkkkkkkk *)

pdw^[1] := pWert^[3];
pdw^[2] := pWert^[2];
pdw^[3] := pWert^[1];

pdw^[0] := INT_TO_BYTE(Kennung);

IF bSendToEmsOnlyIfChanged THEN
	IF (LastdwEMSOut <> dwEMSOut) THEN
		EmsOutFifo(dwEMSOut);
	END_IF
ELSE
	EmsOutFifo(dwEMSOut);
END_IF
LastdwEMSOut := dwEMSOut;
END_FUNCTION_BLOCK

(* POU MdeToEms, ST *)
FUNCTION_BLOCK MdeToEms
VAR_INPUT
 IbsKenn : BYTE;
 MdeKenn : BYTE;
 MdeData : WORD;
END_VAR
VAR
  LastIbsKenn : BYTE;
  LastMdeKenn : BYTE;
  LastMdeData : WORD;
	pbData: POINTER TO ARRAY[0..3] OF BYTE;
	pwData: POINTER TO ARRAY[0..1] OF WORD;
	dwEMSOut: DWORD;
END_VAR
IF (LastIbsKenn <> IbsKenn) OR
   (LastMdeKenn <> MdeKenn) OR
   (LastMdeData <> MdeData) THEN
  LastIbsKenn := IbsKenn;
  LastMdeKenn := MdeKenn;
  LastMdeData := MdeData;

	pbData := ADR( dwEMSOut);
	pwData := ADR( dwEMSOut);
	
	pbData^[0] := IbsKenn;
	pbData^[1] := MdeKenn;
	pwData^[1] := MdeData;
	
	EmsOutFifo( dwEMSOut);
END_IF
END_FUNCTION_BLOCK

(* POU StackFromEms, ST *)
FUNCTION StackFromEms : tEMS_STACK_DATA
VAR_INPUT
	dwEMSIn: DWORD;
END_VAR
VAR
	pdw		: POINTER TO ARRAY[0..3] OF BYTE;
END_VAR
pdw := ADR( dwEMSIn);

StackFromEms.kenn := pdw^[1] AND 16#3F;
StackFromEms.nr := pdw^[2];
StackFromEms.data := pdw^[3];
StackFromEms.toggle := SHR( pdw^[1], 6);
END_FUNCTION

(* POU StackToEms, ST *)
FUNCTION_BLOCK StackToEms
VAR_INPUT
	Data:tEMS_STACK_DATA;
END_VAR
VAR
	LastData:tEMS_STACK_DATA;
	pdw: POINTER TO ARRAY[0..3] OF BYTE;
	pData: POINTER TO ARRAY[0..3] OF BYTE;
	dwEMSOut: DWORD;
END_VAR
IF (LastData.data <> Data.data) OR
   (LastData.kenn <> Data.kenn) OR
   (LastData.nr <> Data.nr) OR
   (LastData.toggle <> Data.toggle) THEN
	LastData := Data;
	pdw := ADR(dwEMSOut);
	pData := ADR(Data);
	
	pdw^[0] := INT_TO_BYTE(IBSK_STACK_DATA);
	pdw^[1] := INT_TO_BYTE(Data.kenn);
	pdw^[2] := Data.nr;
	pdw^[3] := Data.data;
	
	EmsOutFifo(dwEMSOut);
END_IF
END_FUNCTION_BLOCK

(* POU WarnClearToEms, ST *)
FUNCTION WarnClearToEms:BOOL
VAR_INPUT
	Wert: INT;
END_VAR
VAR
	pdw: POINTER TO ARRAY[0..3] OF BYTE;
	pint: POINTER TO ARRAY[0..1] OF BYTE;
	dwEMSOut: DWORD;
END_VAR
pdw := ADR(dwEMSOut);
pint := ADR(Wert);

pdw^[0] := INT_TO_BYTE(IBSK_WARN_CLEAR);
(*pdw^[1] := 0;*)
pdw^[1] := byToggle;
byToggle := byToggle + 1;
pdw^[2] := pint^[1];
pdw^[3] := pint^[0];

WarnClearToEms := EmsOutFifo(dwEMSOut);
END_FUNCTION

(* POU WarnSetToEms, ST *)
FUNCTION WarnSetToEms:BOOL
VAR_INPUT
	Wert: INT;
END_VAR
VAR
	pdw: POINTER TO ARRAY[0..3] OF BYTE;
	pint: POINTER TO ARRAY[0..1] OF BYTE;
	dwEMSOut: DWORD;
END_VAR
pdw := ADR(dwEMSOut);
pint := ADR(Wert);

pdw^[0] := INT_TO_BYTE(IBSK_WARN_SET);
(*pdw^[1] := 0;*)
pdw^[1] := byToggle;
byToggle := byToggle + 1;
pdw^[2] := pint^[1];
pdw^[3] := pint^[0];

WarnSetToEms := EmsOutFifo(dwEMSOut);
END_FUNCTION

(* Visualisation visEmsBildumschaltung
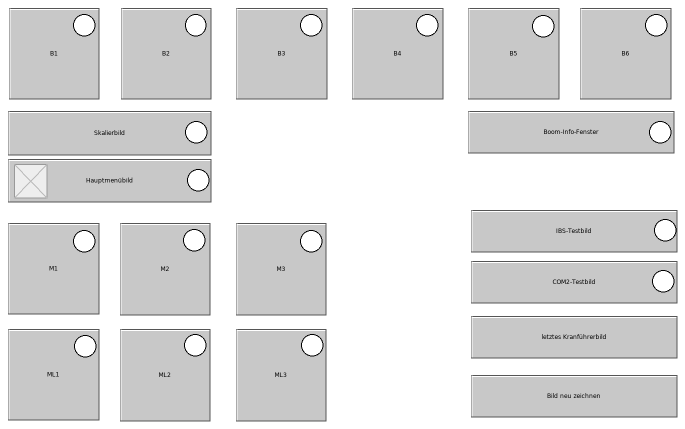
button at (23,15)-(113,106): text "B1"; taps .EmsBild[1]
button at (135,15)-(225,106): text "B2"; taps .EmsBild[2]
button at (250,15)-(341,106): text "B3"; taps .EmsBild[3]
button at (366,15)-(457,106): text "B4"; taps .EmsBild[4]
button at (482,15)-(573,106): text "B5"; taps .EmsBild[28]
button at (594,15)-(685,106): text "B6"; taps .EmsBild[29]
button at (22,230)-(113,321): text "M1"; taps .EmsBild[11]
button at (134,230)-(224,322): text "M2"; taps .EmsBild[12]
button at (250,230)-(340,322): text "M3"; taps .EmsBild[13]
button at (22,118)-(225,162): text "Skalierbild"; taps .EmsBild[5]
ellipse at (87,21)-(109,43): alarm colour if .iEmsAktBild=1
ellipse at (199,21)-(220,43): alarm colour if .iEmsAktBild=2
ellipse at (314,21)-(336,43): alarm colour if .iEmsAktBild=3
ellipse at (430,21)-(452,43): alarm colour if .iEmsAktBild=4
ellipse at (546,22)-(568,44): alarm colour if .iEmsAktBild=28
ellipse at (659,21)-(681,43): alarm colour if .iEmsAktBild=29
button at (22,166)-(225,209): text "Hauptmenübild"; taps .EmsBild[6]
button at (22,336)-(113,427): text "ML1"; taps .EmsBild[14]
button at (134,336)-(224,428): text "ML2"; taps .EmsBild[15]
button at (250,336)-(340,428): text "ML3"; taps .EmsBild[16]
button at (485,323)-(691,365): text "letztes Kranführerbild"; taps .EmsBild[19]
button at (485,382)-(691,424): text "Bild neu zeichnen"; taps .EmsBild[19]
button at (485,217)-(691,259): text "IBS-Testbild"; taps .EmsBild[27]
button at (482,118)-(688,160): text "Boom-Info-Fenster"; taps .EmsBild[30]
button at (485,268)-(691,310): text "COM2-Testbild"; taps .EmsBild[10]
ellipse at (199,128)-(221,150): alarm colour if .iEmsAktBild=5
ellipse at (201,176)-(223,198): alarm colour if .iEmsAktBild=6
ellipse at (87,237)-(109,259): alarm colour if .iEmsAktBild=11
ellipse at (197,236)-(219,258): alarm colour if .iEmsAktBild=12
ellipse at (314,237)-(336,259): alarm colour if .iEmsAktBild=13
ellipse at (88,342)-(110,364): alarm colour if .iEmsAktBild=14
ellipse at (198,341)-(220,363): alarm colour if .iEmsAktBild=15
ellipse at (315,341)-(337,363): alarm colour if .iEmsAktBild=16
ellipse at (668,226)-(690,248): alarm colour if .iEmsAktBild=27
ellipse at (666,277)-(688,299): alarm colour if .iEmsAktBild=10
ellipse at (663,128)-(685,150): alarm colour if .iEmsAktBild=30
bitmap at (28,171)-(61,205): SCHLUESSEL.BMP
*)
